// TIA Portal V19 export
TYPE "C501_STU_KLG_TYPIC"
   STRUCT
      CMD { ExternalAccessible := 'False'; ExternalVisible := 'False'; ExternalWritable := 'False'} : USInt;   // Sturing klep
   END_STRUCT;
END_TYPE
